  	 11:CASE GVL.mb_Output_Registers[GVL.WATERHARDWARETYPE] OF
(* 		GVL.SWPWTR_TIME:
			//GVL.mb_Output_Registers[GVL.REALTIME_PLC_A2D] :=	0;	//nothing to read with FB circuit, just move motor
			IF GVL.mb_Output_Coils[GVL.REALTIME_ADVANCE] THEN		//move the motor forward
				IF TRUE THEN							//test the FB for limit - can't do this, pass through
					GVL_IO.WaterMotorFwd[FTN1] := TRUE;				// turn on the advance output
					GVL_IO.WaterMotorRvs[FTN1] := FALSE;
					wCycleCount := wCycleCount + 1;
					IF wCycleCount > wMotorTimeOn THEN				//done with timer?
						GVL_IO.WaterMotorFwd[FTN1] := FALSE;		//turn off outputs
						GVL_IO.WaterMotorRvs[FTN1] := FALSE;
						GVL.mb_Output_Coils[GVL.REALTIME_ADVANCE] := FALSE; // reset the advance boolean
						wCycleCount := 0;					//reset the timer counter						
					END_IF
				END_IF
			END_IF
			IF GVL.mb_Output_Coils[GVL.REALTIME_RETARD] THEN
				IF TRUE THEN							//test the FB for limit - can't do this, pass through
					GVL_IO.WaterMotorFwd[FTN1] := FALSE;				// turn on the reverse output
					GVL_IO.WaterMotorRvs[FTN1] := TRUE;
					wCycleCount := wCycleCount + 1;
					IF wCycleCount > wMotorTimeOn THEN				//done with timer?
						GVL_IO.WaterMotorFwd[FTN1] := FALSE;		//turn off outputs
						GVL_IO.WaterMotorRvs[FTN1] := FALSE;
						GVL.mb_Output_Coils[GVL.REALTIME_RETARD] := FALSE; // reset the reverse boolean
						wCycleCount := 0;					//reset the timer counter						
					END_IF
				END_IF
			END_IF
		GVL.SWPWTR_FB:
			GVL.mb_Output_Registers[GVL.REALTIME_PLC_A2D] :=	INT_TO_WORD(GVL_IO.WaterInput[FTN1]);
			IF GVL.mb_Output_Coils[GVL.REALTIME_ADVANCE] THEN		//move the motor forward
				IF GVL_IO.WaterInput[FTN1] < 32000 THEN				//test the FB for limit - assumes 32767 is max of 10 VDC
					GVL_IO.WaterMotorFwd[FTN1] := TRUE;				// turn on the advance output
					GVL_IO.WaterMotorRvs[FTN1] := FALSE;
					wCycleCount := wCycleCount + 1;
					IF wCycleCount > wMotorTimeOn THEN				//done with timer?
						GVL_IO.WaterMotorFwd[FTN1] := FALSE;		//turn off outputs
						GVL_IO.WaterMotorRvs[FTN1] := FALSE;
						GVL.mb_Output_Coils[GVL.REALTIME_ADVANCE] := FALSE; // reset the advance boolean
						wCycleCount := 0;					//reset the timer counter						
						//  curr % sweep   curr ticks - min tick allowed      max sweep %            max ticks allowed      min ticks allowed
						GVL.mb_Output_Registers[GVL.SWEEPTRIMONPRESS + (FTN1 * GVL.WORDRUNTIMEGROUPSIZE)]	:= (INT_TO_WORD(GVL_IO.InkInput[FTN1]) - GVL.w_InkInputIntMin[FTN1]) * 
								(GVL.mb_Output_Registers[GVL.MAXSWEEPTRIM]+1) / (GVL.w_InkInputIntMax[FTN1] - GVL.w_InkInputIntMin[FTN1]);
						//need the onpress setting pointed to the current % sweep of the positioner
					END_IF
				END_IF
			END_IF
			IF GVL.mb_Output_Coils[GVL.REALTIME_RETARD] THEN
				IF GVL_IO.WaterInput[FTN1] > 800 THEN				//test the FB for limit - assumes 32767 is max of 10 VDC
					GVL_IO.WaterMotorFwd[FTN1] := FALSE;				// turn on the reverse output
					GVL_IO.WaterMotorRvs[FTN1] := TRUE;
					wCycleCount := wCycleCount + 1;
					IF wCycleCount > wMotorTimeOn THEN				//done with timer?
						GVL_IO.WaterMotorFwd[FTN1] := FALSE;		//turn off outputs
						GVL_IO.WaterMotorRvs[FTN1] := FALSE;
						GVL.mb_Output_Coils[GVL.REALTIME_RETARD] := FALSE; // reset the reverse boolean
						wCycleCount := 0;					//reset the timer counter						
						//  curr % sweep   curr ticks - min tick allowed      max sweep %            max ticks allowed      min ticks allowed
						GVL.mb_Output_Registers[GVL.SWEEPTRIMONPRESS + (FTN1 * GVL.WORDRUNTIMEGROUPSIZE)]	:= (INT_TO_WORD(GVL_IO.InkInput[FTN1]) - GVL.w_InkInputIntMin[FTN1]) * 
								(GVL.mb_Output_Registers[GVL.MAXSWEEPTRIM]+1) / (GVL.w_InkInputIntMax[FTN1] - GVL.w_InkInputIntMin[FTN1]);
						//need the onpress setting pointed to the current % sweep of the positioner
					END_IF
				END_IF
			END_IF
		GVL.SWPWTR_OUTPUT:
			IF( GVL.b_DINTInput) THEN									//how big should the adv / ret control increment be?
				w_output_incr :=  DINT_TO_INT(GVL.d_DINT10V / 100);
			ELSE
				w_output_incr := (GVL.i_INT10V / 100);
			END_IF
			GVL.mb_Output_Registers[GVL.REALTIME_PLC_A2D] :=	INT_TO_WORD(GVL_IO.WaterSweepOut[FTN1]);
			IF GVL.mb_Output_Coils[GVL.REALTIME_ADVANCE] THEN
				IF GVL_IO.WaterSweepOut[FTN1] < (w_output_incr * 10) THEN
					GVL_IO.WaterSweepOut[FTN1] := GVL_IO.WaterSweepOut[FTN1] + w_output_incr;
				END_IF
				GVL.mb_Output_Coils[GVL.REALTIME_ADVANCE] := FALSE;
			END_IF
			IF GVL.mb_Output_Coils[GVL.REALTIME_RETARD] THEN
				IF GVL_IO.WaterSweepOut[FTN1] > w_output_incr THEN
					GVL_IO.WaterSweepOut[FTN1] := GVL_IO.WaterSweepOut[FTN1] - w_output_incr;
				END_IF
				GVL.mb_Output_Coils[GVL.REALTIME_RETARD] := FALSE;
			END_IF			
 *)
		GVL.SWPWTR_BRIDGE:
		END_CASE
	 12:CASE GVL.mb_Output_Registers[GVL.WATERHARDWARETYPE] OF
(* 		GVL.SWPWTR_TIME:
			//GVL.mb_Output_Registers[GVL.REALTIME_PLC_A2D] :=	0;	//nothing to read with FB circuit, just move motor
			IF GVL.mb_Output_Coils[GVL.REALTIME_ADVANCE] THEN		//move the motor forward
				IF TRUE THEN							//test the FB for limit - can't do this, pass through
					GVL_IO.WaterMotorFwd[FTN2] := TRUE;				// turn on the advance output
					GVL_IO.WaterMotorRvs[FTN2] := FALSE;
					wCycleCount := wCycleCount + 1;
					IF wCycleCount > wMotorTimeOn THEN				//done with timer?
						GVL_IO.WaterMotorFwd[FTN2] := FALSE;		//turn off outputs
						GVL_IO.WaterMotorRvs[FTN2] := FALSE;
						GVL.mb_Output_Coils[GVL.REALTIME_ADVANCE] := FALSE; // reset the advance boolean
						wCycleCount := 0;					//reset the timer counter						
					END_IF
				END_IF
			END_IF
			IF GVL.mb_Output_Coils[GVL.REALTIME_RETARD] THEN
				IF TRUE THEN							//test the FB for limit - can't do this, pass through
					GVL_IO.WaterMotorFwd[FTN2] := FALSE;				// turn on the reverse output
					GVL_IO.WaterMotorRvs[FTN2] := TRUE;
					wCycleCount := wCycleCount + 1;
					IF wCycleCount > wMotorTimeOn THEN				//done with timer?
						GVL_IO.WaterMotorFwd[FTN2] := FALSE;		//turn off outputs
						GVL_IO.WaterMotorRvs[FTN2] := FALSE;
						GVL.mb_Output_Coils[GVL.REALTIME_RETARD] := FALSE; // reset the reverse boolean
						wCycleCount := 0;					//reset the timer counter						
					END_IF
				END_IF
			END_IF
		GVL.SWPWTR_FB:
			GVL.mb_Output_Registers[GVL.REALTIME_PLC_A2D] :=	INT_TO_WORD(GVL_IO.WaterInput[FTN2]);
			IF GVL.mb_Output_Coils[GVL.REALTIME_ADVANCE] THEN		//move the motor forward
				IF GVL_IO.WaterInput[FTN2] < 32000 THEN				//test the FB for limit - assumes 32767 is max of 10 VDC
					GVL_IO.WaterMotorFwd[FTN2] := TRUE;				// turn on the advance output
					GVL_IO.WaterMotorRvs[FTN2] := FALSE;
					wCycleCount := wCycleCount + 1;
					IF wCycleCount > wMotorTimeOn THEN				//done with timer?
						GVL_IO.WaterMotorFwd[FTN2] := FALSE;		//turn off outputs
						GVL_IO.WaterMotorRvs[FTN2] := FALSE;
						GVL.mb_Output_Coils[GVL.REALTIME_ADVANCE] := FALSE; // reset the advance boolean
						wCycleCount := 0;					//reset the timer counter						
						//  curr % sweep   curr ticks - min tick allowed      max sweep %            max ticks allowed      min ticks allowed
						GVL.mb_Output_Registers[GVL.SWEEPTRIMONPRESS + (FTN2 * GVL.WORDRUNTIMEGROUPSIZE)]	:= (INT_TO_WORD(GVL_IO.InkInput[FTN2]) - GVL.w_InkInputIntMin[FTN2]) * 
								(GVL.mb_Output_Registers[GVL.MAXSWEEPTRIM]+1) / (GVL.w_InkInputIntMax[FTN2] - GVL.w_InkInputIntMin[FTN2]);
						//need the onpress setting pointed to the current % sweep of the positioner
					END_IF
				END_IF
			END_IF
			IF GVL.mb_Output_Coils[GVL.REALTIME_RETARD] THEN
				IF GVL_IO.WaterInput[FTN2] > 800 THEN				//test the FB for limit - assumes 32767 is max of 10 VDC
					GVL_IO.WaterMotorFwd[FTN2] := FALSE;				// turn on the reverse output
					GVL_IO.WaterMotorRvs[FTN2] := TRUE;
					wCycleCount := wCycleCount + 1;
					IF wCycleCount > wMotorTimeOn THEN				//done with timer?
						GVL_IO.WaterMotorFwd[FTN2] := FALSE;		//turn off outputs
						GVL_IO.WaterMotorRvs[FTN2] := FALSE;
						GVL.mb_Output_Coils[GVL.REALTIME_RETARD] := FALSE; // reset the reverse boolean
						wCycleCount := 0;					//reset the timer counter						
						//  curr % sweep   curr ticks - min tick allowed      max sweep %            max ticks allowed      min ticks allowed
						GVL.mb_Output_Registers[GVL.SWEEPTRIMONPRESS + (FTN2 * GVL.WORDRUNTIMEGROUPSIZE)]	:= (INT_TO_WORD(GVL_IO.InkInput[FTN2]) - GVL.w_InkInputIntMin[FTN2]) * 
								(GVL.mb_Output_Registers[GVL.MAXSWEEPTRIM]+1) / (GVL.w_InkInputIntMax[FTN2] - GVL.w_InkInputIntMin[FTN2]);
						//need the onpress setting pointed to the current % sweep of the positioner
					END_IF
				END_IF
			END_IF
		GVL.SWPWTR_OUTPUT:
			IF( GVL.b_DINTInput) THEN									//how big should the adv / ret control increment be?
				w_output_incr :=  DINT_TO_INT(GVL.d_DINT10V / 100);
			ELSE
				w_output_incr := (GVL.i_INT10V / 100);
			END_IF
			GVL.mb_Output_Registers[GVL.REALTIME_PLC_A2D] :=	INT_TO_WORD(GVL_IO.WaterSweepOut[FTN2]);
			IF GVL.mb_Output_Coils[GVL.REALTIME_ADVANCE] THEN
				IF GVL_IO.WaterSweepOut[FTN2] < (w_output_incr * 10) THEN
					GVL_IO.WaterSweepOut[FTN2] := GVL_IO.WaterSweepOut[FTN2] + w_output_incr;
				END_IF
				GVL.mb_Output_Coils[GVL.REALTIME_ADVANCE] := FALSE;
			END_IF
			IF GVL.mb_Output_Coils[GVL.REALTIME_RETARD] THEN
				IF GVL_IO.WaterSweepOut[FTN2] > w_output_incr THEN
					GVL_IO.WaterSweepOut[FTN2] := GVL_IO.WaterSweepOut[FTN2] - w_output_incr;
				END_IF
				GVL.mb_Output_Coils[GVL.REALTIME_RETARD] := FALSE;
			END_IF			
 *)
		GVL.SWPWTR_BRIDGE:
		END_CASE
	 13:CASE GVL.mb_Output_Registers[GVL.WATERHARDWARETYPE] OF
(* 		GVL.SWPWTR_TIME:
			//GVL.mb_Output_Registers[GVL.REALTIME_PLC_A2D] :=	0;	//nothing to read with FB circuit, just move motor
			IF GVL.mb_Output_Coils[GVL.REALTIME_ADVANCE] THEN		//move the motor forward
				IF TRUE THEN							//test the FB for limit - can't do this, pass through
					GVL_IO.WaterMotorFwd[FTN3] := TRUE;				// turn on the advance output
					GVL_IO.WaterMotorRvs[FTN3] := FALSE;
					wCycleCount := wCycleCount + 1;
					IF wCycleCount > wMotorTimeOn THEN				//done with timer?
						GVL_IO.WaterMotorFwd[FTN3] := FALSE;		//turn off outputs
						GVL_IO.WaterMotorRvs[FTN3] := FALSE;
						GVL.mb_Output_Coils[GVL.REALTIME_ADVANCE] := FALSE; // reset the advance boolean
						wCycleCount := 0;					//reset the timer counter						
					END_IF
				END_IF
			END_IF
			IF GVL.mb_Output_Coils[GVL.REALTIME_RETARD] THEN
				IF TRUE THEN							//test the FB for limit - can't do this, pass through
					GVL_IO.WaterMotorFwd[FTN3] := FALSE;				// turn on the reverse output
					GVL_IO.WaterMotorRvs[FTN3] := TRUE;
					wCycleCount := wCycleCount + 1;
					IF wCycleCount > wMotorTimeOn THEN				//done with timer?
						GVL_IO.WaterMotorFwd[FTN3] := FALSE;		//turn off outputs
						GVL_IO.WaterMotorRvs[FTN3] := FALSE;
						GVL.mb_Output_Coils[GVL.REALTIME_RETARD] := FALSE; // reset the reverse boolean
						wCycleCount := 0;					//reset the timer counter						
					END_IF
				END_IF
			END_IF
		GVL.SWPWTR_FB:
			GVL.mb_Output_Registers[GVL.REALTIME_PLC_A2D] :=	INT_TO_WORD(GVL_IO.WaterInput[FTN3]);
			IF GVL.mb_Output_Coils[GVL.REALTIME_ADVANCE] THEN		//move the motor forward
				IF GVL_IO.WaterInput[FTN3] < 32000 THEN				//test the FB for limit - assumes 32767 is max of 10 VDC
					GVL_IO.WaterMotorFwd[FTN3] := TRUE;				// turn on the advance output
					GVL_IO.WaterMotorRvs[FTN3] := FALSE;
					wCycleCount := wCycleCount + 1;
					IF wCycleCount > wMotorTimeOn THEN				//done with timer?
						GVL_IO.WaterMotorFwd[FTN3] := FALSE;		//turn off outputs
						GVL_IO.WaterMotorRvs[FTN3] := FALSE;
						GVL.mb_Output_Coils[GVL.REALTIME_ADVANCE] := FALSE; // reset the advance boolean
						wCycleCount := 0;					//reset the timer counter						
						//  curr % sweep   curr ticks - min tick allowed      max sweep %            max ticks allowed      min ticks allowed
						GVL.mb_Output_Registers[GVL.SWEEPTRIMONPRESS + (FTN3 * GVL.WORDRUNTIMEGROUPSIZE)]	:= (INT_TO_WORD(GVL_IO.InkInput[FTN3]) - GVL.w_InkInputIntMin[FTN3]) * 
								(GVL.mb_Output_Registers[GVL.MAXSWEEPTRIM]+1) / (GVL.w_InkInputIntMax[FTN3] - GVL.w_InkInputIntMin[FTN3]);
						//need the onpress setting pointed to the current % sweep of the positioner
					END_IF
				END_IF
			END_IF
			IF GVL.mb_Output_Coils[GVL.REALTIME_RETARD] THEN
				IF GVL_IO.WaterInput[FTN3] > 800 THEN				//test the FB for limit - assumes 32767 is max of 10 VDC
					GVL_IO.WaterMotorFwd[FTN3] := FALSE;				// turn on the reverse output
					GVL_IO.WaterMotorRvs[FTN3] := TRUE;
					wCycleCount := wCycleCount + 1;
					IF wCycleCount > wMotorTimeOn THEN				//done with timer?
						GVL_IO.WaterMotorFwd[FTN3] := FALSE;		//turn off outputs
						GVL_IO.WaterMotorRvs[FTN3] := FALSE;
						GVL.mb_Output_Coils[GVL.REALTIME_RETARD] := FALSE; // reset the reverse boolean
						wCycleCount := 0;					//reset the timer counter						
						//  curr % sweep   curr ticks - min tick allowed      max sweep %            max ticks allowed      min ticks allowed
						GVL.mb_Output_Registers[GVL.SWEEPTRIMONPRESS + (FTN3 * GVL.WORDRUNTIMEGROUPSIZE)]	:= (INT_TO_WORD(GVL_IO.InkInput[FTN3]) - GVL.w_InkInputIntMin[FTN3]) * 
								(GVL.mb_Output_Registers[GVL.MAXSWEEPTRIM]+1) / (GVL.w_InkInputIntMax[FTN3] - GVL.w_InkInputIntMin[FTN3]);
						//need the onpress setting pointed to the current % sweep of the positioner
					END_IF
				END_IF
			END_IF
		GVL.SWPWTR_OUTPUT:
			IF( GVL.b_DINTInput) THEN									//how big should the adv / ret control increment be?
				w_output_incr :=  DINT_TO_INT(GVL.d_DINT10V / 100);
			ELSE
				w_output_incr := (GVL.i_INT10V / 100);
			END_IF
			GVL.mb_Output_Registers[GVL.REALTIME_PLC_A2D] :=	INT_TO_WORD(GVL_IO.WaterSweepOut[FTN3]);
			IF GVL.mb_Output_Coils[GVL.REALTIME_ADVANCE] THEN
				IF GVL_IO.WaterSweepOut[FTN3] < (w_output_incr * 10) THEN
					GVL_IO.WaterSweepOut[FTN3] := GVL_IO.WaterSweepOut[FTN3] + w_output_incr;
				END_IF
				GVL.mb_Output_Coils[GVL.REALTIME_ADVANCE] := FALSE;
			END_IF
			IF GVL.mb_Output_Coils[GVL.REALTIME_RETARD] THEN
				IF GVL_IO.WaterSweepOut[FTN3] > w_output_incr THEN
					GVL_IO.WaterSweepOut[FTN3] := GVL_IO.WaterSweepOut[FTN3] - w_output_incr;
				END_IF
				GVL.mb_Output_Coils[GVL.REALTIME_RETARD] := FALSE;
			END_IF			
 *)
		GVL.SWPWTR_BRIDGE:
		END_CASE
	 14:CASE GVL.mb_Output_Registers[GVL.WATERHARDWARETYPE] OF
(* 		GVL.SWPWTR_TIME:
			//GVL.mb_Output_Registers[GVL.REALTIME_PLC_A2D] :=	0;	//nothing to read with FB circuit, just move motor
			IF GVL.mb_Output_Coils[GVL.REALTIME_ADVANCE] THEN		//move the motor forward
				IF TRUE THEN							//test the FB for limit - can't do this, pass through
					GVL_IO.WaterMotorFwd[FTN4] := TRUE;				// turn on the advance output
					GVL_IO.WaterMotorRvs[FTN4] := FALSE;
					wCycleCount := wCycleCount + 1;
					IF wCycleCount > wMotorTimeOn THEN				//done with timer?
						GVL_IO.WaterMotorFwd[FTN4] := FALSE;		//turn off outputs
						GVL_IO.WaterMotorRvs[FTN4] := FALSE;
						GVL.mb_Output_Coils[GVL.REALTIME_ADVANCE] := FALSE; // reset the advance boolean
						wCycleCount := 0;					//reset the timer counter						
					END_IF
				END_IF
			END_IF
			IF GVL.mb_Output_Coils[GVL.REALTIME_RETARD] THEN
				IF TRUE THEN							//test the FB for limit - can't do this, pass through
					GVL_IO.WaterMotorFwd[FTN4] := FALSE;				// turn on the reverse output
					GVL_IO.WaterMotorRvs[FTN4] := TRUE;
					wCycleCount := wCycleCount + 1;
					IF wCycleCount > wMotorTimeOn THEN				//done with timer?
						GVL_IO.WaterMotorFwd[FTN4] := FALSE;		//turn off outputs
						GVL_IO.WaterMotorRvs[FTN4] := FALSE;
						GVL.mb_Output_Coils[GVL.REALTIME_RETARD] := FALSE; // reset the reverse boolean
						wCycleCount := 0;					//reset the timer counter						
					END_IF
				END_IF
			END_IF
		GVL.SWPWTR_FB:
			GVL.mb_Output_Registers[GVL.REALTIME_PLC_A2D] :=	INT_TO_WORD(GVL_IO.WaterInput[FTN4]);
			IF GVL.mb_Output_Coils[GVL.REALTIME_ADVANCE] THEN		//move the motor forward
				IF GVL_IO.WaterInput[FTN4] < 32000 THEN				//test the FB for limit - assumes 32767 is max of 10 VDC
					GVL_IO.WaterMotorFwd[FTN4] := TRUE;				// turn on the advance output
					GVL_IO.WaterMotorRvs[FTN4] := FALSE;
					wCycleCount := wCycleCount + 1;
					IF wCycleCount > wMotorTimeOn THEN				//done with timer?
						GVL_IO.WaterMotorFwd[FTN4] := FALSE;		//turn off outputs
						GVL_IO.WaterMotorRvs[FTN4] := FALSE;
						GVL.mb_Output_Coils[GVL.REALTIME_ADVANCE] := FALSE; // reset the advance boolean
						wCycleCount := 0;					//reset the timer counter						
						//  curr % sweep   curr ticks - min tick allowed      max sweep %            max ticks allowed      min ticks allowed
						GVL.mb_Output_Registers[GVL.SWEEPTRIMONPRESS + (FTN4 * GVL.WORDRUNTIMEGROUPSIZE)]	:= (INT_TO_WORD(GVL_IO.InkInput[FTN4]) - GVL.w_InkInputIntMin[FTN4]) * 
								(GVL.mb_Output_Registers[GVL.MAXSWEEPTRIM]+1) / (GVL.w_InkInputIntMax[FTN4] - GVL.w_InkInputIntMin[FTN4]);
						//need the onpress setting pointed to the current % sweep of the positioner
					END_IF
				END_IF
			END_IF
			IF GVL.mb_Output_Coils[GVL.REALTIME_RETARD] THEN
				IF GVL_IO.WaterInput[FTN4] > 800 THEN				//test the FB for limit - assumes 32767 is max of 10 VDC
					GVL_IO.WaterMotorFwd[FTN4] := FALSE;				// turn on the reverse output
					GVL_IO.WaterMotorRvs[FTN4] := TRUE;
					wCycleCount := wCycleCount + 1;
					IF wCycleCount > wMotorTimeOn THEN				//done with timer?
						GVL_IO.WaterMotorFwd[FTN4] := FALSE;		//turn off outputs
						GVL_IO.WaterMotorRvs[FTN4] := FALSE;
						GVL.mb_Output_Coils[GVL.REALTIME_RETARD] := FALSE; // reset the reverse boolean
						wCycleCount := 0;					//reset the timer counter						
						//  curr % sweep   curr ticks - min tick allowed      max sweep %            max ticks allowed      min ticks allowed
						GVL.mb_Output_Registers[GVL.SWEEPTRIMONPRESS + (FTN4 * GVL.WORDRUNTIMEGROUPSIZE)]	:= (INT_TO_WORD(GVL_IO.InkInput[FTN4]) - GVL.w_InkInputIntMin[FTN4]) * 
								(GVL.mb_Output_Registers[GVL.MAXSWEEPTRIM]+1) / (GVL.w_InkInputIntMax[FTN4] - GVL.w_InkInputIntMin[FTN4]);
						//need the onpress setting pointed to the current % sweep of the positioner
					END_IF
				END_IF
			END_IF
		GVL.SWPWTR_OUTPUT:
			IF( GVL.b_DINTInput) THEN									//how big should the adv / ret control increment be?
				w_output_incr :=  DINT_TO_INT(GVL.d_DINT10V / 100);
			ELSE
				w_output_incr := (GVL.i_INT10V / 100);
			END_IF
			GVL.mb_Output_Registers[GVL.REALTIME_PLC_A2D] :=	INT_TO_WORD(GVL_IO.WaterSweepOut[FTN4]);
			IF GVL.mb_Output_Coils[GVL.REALTIME_ADVANCE] THEN
				IF GVL_IO.WaterSweepOut[FTN4] < (w_output_incr * 10) THEN
					GVL_IO.WaterSweepOut[FTN4] := GVL_IO.WaterSweepOut[FTN4] + w_output_incr;
				END_IF
				GVL.mb_Output_Coils[GVL.REALTIME_ADVANCE] := FALSE;
			END_IF
			IF GVL.mb_Output_Coils[GVL.REALTIME_RETARD] THEN
				IF GVL_IO.WaterSweepOut[FTN4] > w_output_incr THEN
					GVL_IO.WaterSweepOut[FTN4] := GVL_IO.WaterSweepOut[FTN4] - w_output_incr;
				END_IF
				GVL.mb_Output_Coils[GVL.REALTIME_RETARD] := FALSE;
			END_IF			
 *)
		GVL.SWPWTR_BRIDGE:
		END_CASE
	 15:CASE GVL.mb_Output_Registers[GVL.WATERHARDWARETYPE] OF
(* 		GVL.SWPWTR_TIME:
			//GVL.mb_Output_Registers[GVL.REALTIME_PLC_A2D] :=	0;	//nothing to read with FB circuit, just move motor
			IF GVL.mb_Output_Coils[GVL.REALTIME_ADVANCE] THEN		//move the motor forward
				IF TRUE THEN							//test the FB for limit - can't do this, pass through
					GVL_IO.WaterMotorFwd[FTN5] := TRUE;				// turn on the advance output
					GVL_IO.WaterMotorRvs[FTN5] := FALSE;
					wCycleCount := wCycleCount + 1;
					IF wCycleCount > wMotorTimeOn THEN				//done with timer?
						GVL_IO.WaterMotorFwd[FTN5] := FALSE;		//turn off outputs
						GVL_IO.WaterMotorRvs[FTN5] := FALSE;
						GVL.mb_Output_Coils[GVL.REALTIME_ADVANCE] := FALSE; // reset the advance boolean
						wCycleCount := 0;					//reset the timer counter						
					END_IF
				END_IF
			END_IF
			IF GVL.mb_Output_Coils[GVL.REALTIME_RETARD] THEN
				IF TRUE THEN							//test the FB for limit - can't do this, pass through
					GVL_IO.WaterMotorFwd[FTN5] := FALSE;				// turn on the reverse output
					GVL_IO.WaterMotorRvs[FTN5] := TRUE;
					wCycleCount := wCycleCount + 1;
					IF wCycleCount > wMotorTimeOn THEN				//done with timer?
						GVL_IO.WaterMotorFwd[FTN5] := FALSE;		//turn off outputs
						GVL_IO.WaterMotorRvs[FTN5] := FALSE;
						GVL.mb_Output_Coils[GVL.REALTIME_RETARD] := FALSE; // reset the reverse boolean
						wCycleCount := 0;					//reset the timer counter						
					END_IF
				END_IF
			END_IF
		GVL.SWPWTR_FB:
			GVL.mb_Output_Registers[GVL.REALTIME_PLC_A2D] :=	INT_TO_WORD(GVL_IO.WaterInput[FTN5]);
			IF GVL.mb_Output_Coils[GVL.REALTIME_ADVANCE] THEN		//move the motor forward
				IF GVL_IO.WaterInput[FTN5] < 32000 THEN				//test the FB for limit - assumes 32767 is max of 10 VDC
					GVL_IO.WaterMotorFwd[FTN5] := TRUE;				// turn on the advance output
					GVL_IO.WaterMotorRvs[FTN5] := FALSE;
					wCycleCount := wCycleCount + 1;
					IF wCycleCount > wMotorTimeOn THEN				//done with timer?
						GVL_IO.WaterMotorFwd[FTN5] := FALSE;		//turn off outputs
						GVL_IO.WaterMotorRvs[FTN5] := FALSE;
						GVL.mb_Output_Coils[GVL.REALTIME_ADVANCE] := FALSE; // reset the advance boolean
						wCycleCount := 0;					//reset the timer counter						
						//  curr % sweep   curr ticks - min tick allowed      max sweep %            max ticks allowed      min ticks allowed
						GVL.mb_Output_Registers[GVL.SWEEPTRIMONPRESS + (FTN5 * GVL.WORDRUNTIMEGROUPSIZE)]	:= (INT_TO_WORD(GVL_IO.InkInput[FTN5]) - GVL.w_InkInputIntMin[FTN5]) * 
								(GVL.mb_Output_Registers[GVL.MAXSWEEPTRIM]+1) / (GVL.w_InkInputIntMax[FTN5] - GVL.w_InkInputIntMin[FTN5]);
						//need the onpress setting pointed to the current % sweep of the positioner
					END_IF
				END_IF
			END_IF
			IF GVL.mb_Output_Coils[GVL.REALTIME_RETARD] THEN
				IF GVL_IO.WaterInput[FTN5] > 800 THEN				//test the FB for limit - assumes 32767 is max of 10 VDC
					GVL_IO.WaterMotorFwd[FTN5] := FALSE;				// turn on the reverse output
					GVL_IO.WaterMotorRvs[FTN5] := TRUE;
					wCycleCount := wCycleCount + 1;
					IF wCycleCount > wMotorTimeOn THEN				//done with timer?
						GVL_IO.WaterMotorFwd[FTN5] := FALSE;		//turn off outputs
						GVL_IO.WaterMotorRvs[FTN5] := FALSE;
						GVL.mb_Output_Coils[GVL.REALTIME_RETARD] := FALSE; // reset the reverse boolean
						wCycleCount := 0;					//reset the timer counter						
						//  curr % sweep   curr ticks - min tick allowed      max sweep %            max ticks allowed      min ticks allowed
						GVL.mb_Output_Registers[GVL.SWEEPTRIMONPRESS + (FTN5 * GVL.WORDRUNTIMEGROUPSIZE)]	:= (INT_TO_WORD(GVL_IO.InkInput[FTN5]) - GVL.w_InkInputIntMin[FTN5]) * 
								(GVL.mb_Output_Registers[GVL.MAXSWEEPTRIM]+1) / (GVL.w_InkInputIntMax[FTN5] - GVL.w_InkInputIntMin[FTN5]);
						//need the onpress setting pointed to the current % sweep of the positioner
					END_IF
				END_IF
			END_IF
		GVL.SWPWTR_OUTPUT:
			IF( GVL.b_DINTInput) THEN									//how big should the adv / ret control increment be?
				w_output_incr :=  DINT_TO_INT(GVL.d_DINT10V / 100);
			ELSE
				w_output_incr := (GVL.i_INT10V / 100);
			END_IF
			GVL.mb_Output_Registers[GVL.REALTIME_PLC_A2D] :=	INT_TO_WORD(GVL_IO.WaterSweepOut[FTN5]);
			IF GVL.mb_Output_Coils[GVL.REALTIME_ADVANCE] THEN
				IF GVL_IO.WaterSweepOut[FTN5] < (w_output_incr * 10) THEN
					GVL_IO.WaterSweepOut[FTN5] := GVL_IO.WaterSweepOut[FTN5] + w_output_incr;
				END_IF
				GVL.mb_Output_Coils[GVL.REALTIME_ADVANCE] := FALSE;
			END_IF
			IF GVL.mb_Output_Coils[GVL.REALTIME_RETARD] THEN
				IF GVL_IO.WaterSweepOut[FTN5] > w_output_incr THEN
					GVL_IO.WaterSweepOut[FTN5] := GVL_IO.WaterSweepOut[FTN5] - w_output_incr;
				END_IF
				GVL.mb_Output_Coils[GVL.REALTIME_RETARD] := FALSE;
			END_IF			
 *)
		GVL.SWPWTR_BRIDGE:
		END_CASE
	 16:	CASE GVL.mb_Output_Registers[GVL.WATERHARDWARETYPE] OF
(* 		GVL.SWPWTR_TIME:
			//GVL.mb_Output_Registers[GVL.REALTIME_PLC_A2D] :=	0;	//nothing to read with FB circuit, just move motor
			IF GVL.mb_Output_Coils[GVL.REALTIME_ADVANCE] THEN		//move the motor forward
				IF TRUE THEN							//test the FB for limit - can't do this, pass through
					GVL_IO.WaterMotorFwd[FTN6] := TRUE;				// turn on the advance output
					GVL_IO.WaterMotorRvs[FTN6] := FALSE;
					wCycleCount := wCycleCount + 1;
					IF wCycleCount > wMotorTimeOn THEN				//done with timer?
						GVL_IO.WaterMotorFwd[FTN6] := FALSE;		//turn off outputs
						GVL_IO.WaterMotorRvs[FTN6] := FALSE;
						GVL.mb_Output_Coils[GVL.REALTIME_ADVANCE] := FALSE; // reset the advance boolean
						wCycleCount := 0;					//reset the timer counter						
					END_IF
				END_IF
			END_IF
			IF GVL.mb_Output_Coils[GVL.REALTIME_RETARD] THEN
				IF TRUE THEN							//test the FB for limit - can't do this, pass through
					GVL_IO.WaterMotorFwd[FTN6] := FALSE;				// turn on the reverse output
					GVL_IO.WaterMotorRvs[FTN6] := TRUE;
					wCycleCount := wCycleCount + 1;
					IF wCycleCount > wMotorTimeOn THEN				//done with timer?
						GVL_IO.WaterMotorFwd[FTN6] := FALSE;		//turn off outputs
						GVL_IO.WaterMotorRvs[FTN6] := FALSE;
						GVL.mb_Output_Coils[GVL.REALTIME_RETARD] := FALSE; // reset the reverse boolean
						wCycleCount := 0;					//reset the timer counter						
					END_IF
				END_IF
			END_IF
		GVL.SWPWTR_FB:
			GVL.mb_Output_Registers[GVL.REALTIME_PLC_A2D] :=	INT_TO_WORD(GVL_IO.WaterInput[FTN6]);
			IF GVL.mb_Output_Coils[GVL.REALTIME_ADVANCE] THEN		//move the motor forward
				IF GVL_IO.WaterInput[FTN6] < 32000 THEN				//test the FB for limit - assumes 32767 is max of 10 VDC
					GVL_IO.WaterMotorFwd[FTN6] := TRUE;				// turn on the advance output
					GVL_IO.WaterMotorRvs[FTN6] := FALSE;
					wCycleCount := wCycleCount + 1;
					IF wCycleCount > wMotorTimeOn THEN				//done with timer?
						GVL_IO.WaterMotorFwd[FTN6] := FALSE;		//turn off outputs
						GVL_IO.WaterMotorRvs[FTN6] := FALSE;
						GVL.mb_Output_Coils[GVL.REALTIME_ADVANCE] := FALSE; // reset the advance boolean
						wCycleCount := 0;					//reset the timer counter						
						//  curr % sweep   curr ticks - min tick allowed      max sweep %            max ticks allowed      min ticks allowed
						GVL.mb_Output_Registers[GVL.SWEEPTRIMONPRESS + (FTN6 * GVL.WORDRUNTIMEGROUPSIZE)]	:= (INT_TO_WORD(GVL_IO.InkInput[FTN6]) - GVL.w_InkInputIntMin[FTN6]) * 
								(GVL.mb_Output_Registers[GVL.MAXSWEEPTRIM]+1) / (GVL.w_InkInputIntMax[FTN6] - GVL.w_InkInputIntMin[FTN6]);
						//need the onpress setting pointed to the current % sweep of the positioner
					END_IF
				END_IF
			END_IF
			IF GVL.mb_Output_Coils[GVL.REALTIME_RETARD] THEN
				IF GVL_IO.WaterInput[FTN6] > 800 THEN				//test the FB for limit - assumes 32767 is max of 10 VDC
					GVL_IO.WaterMotorFwd[FTN6] := FALSE;				// turn on the reverse output
					GVL_IO.WaterMotorRvs[FTN6] := TRUE;
					wCycleCount := wCycleCount + 1;
					IF wCycleCount > wMotorTimeOn THEN				//done with timer?
						GVL_IO.WaterMotorFwd[FTN6] := FALSE;		//turn off outputs
						GVL_IO.WaterMotorRvs[FTN6] := FALSE;
						GVL.mb_Output_Coils[GVL.REALTIME_RETARD] := FALSE; // reset the reverse boolean
						wCycleCount := 0;					//reset the timer counter						
						//  curr % sweep   curr ticks - min tick allowed      max sweep %            max ticks allowed      min ticks allowed
						GVL.mb_Output_Registers[GVL.SWEEPTRIMONPRESS + (FTN6 * GVL.WORDRUNTIMEGROUPSIZE)]	:= (INT_TO_WORD(GVL_IO.InkInput[FTN6]) - GVL.w_InkInputIntMin[FTN6]) * 
								(GVL.mb_Output_Registers[GVL.MAXSWEEPTRIM]+1) / (GVL.w_InkInputIntMax[FTN6] - GVL.w_InkInputIntMin[FTN6]);
						//need the onpress setting pointed to the current % sweep of the positioner
					END_IF
				END_IF
			END_IF
		GVL.SWPWTR_OUTPUT:
			IF( GVL.b_DINTInput) THEN									//how big should the adv / ret control increment be?
				w_output_incr :=  DINT_TO_INT(GVL.d_DINT10V / 100);
			ELSE
				w_output_incr := (GVL.i_INT10V / 100);
			END_IF
			GVL.mb_Output_Registers[GVL.REALTIME_PLC_A2D] :=	INT_TO_WORD(GVL_IO.WaterSweepOut[FTN6]);
			IF GVL.mb_Output_Coils[GVL.REALTIME_ADVANCE] THEN
				IF GVL_IO.WaterSweepOut[FTN6] < (w_output_incr * 10) THEN
					GVL_IO.WaterSweepOut[FTN6] := GVL_IO.WaterSweepOut[FTN6] + w_output_incr;
				END_IF
				GVL.mb_Output_Coils[GVL.REALTIME_ADVANCE] := FALSE;
			END_IF
			IF GVL.mb_Output_Coils[GVL.REALTIME_RETARD] THEN
				IF GVL_IO.WaterSweepOut[FTN6] > w_output_incr THEN
					GVL_IO.WaterSweepOut[FTN6] := GVL_IO.WaterSweepOut[FTN6] - w_output_incr;
				END_IF
				GVL.mb_Output_Coils[GVL.REALTIME_RETARD] := FALSE;
			END_IF			
 *)
		GVL.SWPWTR_BRIDGE:
		END_CASE
	 17:CASE GVL.mb_Output_Registers[GVL.WATERHARDWARETYPE] OF
(* 		GVL.SWPWTR_TIME:
			//GVL.mb_Output_Registers[GVL.REALTIME_PLC_A2D] :=	0;	//nothing to read with FB circuit, just move motor
			IF GVL.mb_Output_Coils[GVL.REALTIME_ADVANCE] THEN		//move the motor forward
				IF TRUE THEN							//test the FB for limit - can't do this, pass through
					GVL_IO.WaterMotorFwd[FTN7] := TRUE;				// turn on the advance output
					GVL_IO.WaterMotorRvs[FTN7] := FALSE;
					wCycleCount := wCycleCount + 1;
					IF wCycleCount > wMotorTimeOn THEN				//done with timer?
						GVL_IO.WaterMotorFwd[FTN7] := FALSE;		//turn off outputs
						GVL_IO.WaterMotorRvs[FTN7] := FALSE;
						GVL.mb_Output_Coils[GVL.REALTIME_ADVANCE] := FALSE; // reset the advance boolean
						wCycleCount := 0;					//reset the timer counter						
					END_IF
				END_IF
			END_IF
			IF GVL.mb_Output_Coils[GVL.REALTIME_RETARD] THEN
				IF TRUE THEN							//test the FB for limit - can't do this, pass through
					GVL_IO.WaterMotorFwd[FTN7] := FALSE;				// turn on the reverse output
					GVL_IO.WaterMotorRvs[FTN7] := TRUE;
					wCycleCount := wCycleCount + 1;
					IF wCycleCount > wMotorTimeOn THEN				//done with timer?
						GVL_IO.WaterMotorFwd[FTN7] := FALSE;		//turn off outputs
						GVL_IO.WaterMotorRvs[FTN7] := FALSE;
						GVL.mb_Output_Coils[GVL.REALTIME_RETARD] := FALSE; // reset the reverse boolean
						wCycleCount := 0;					//reset the timer counter						
					END_IF
				END_IF
			END_IF
		GVL.SWPWTR_FB:
			GVL.mb_Output_Registers[GVL.REALTIME_PLC_A2D] :=	INT_TO_WORD(GVL_IO.WaterInput[FTN7]);
			IF GVL.mb_Output_Coils[GVL.REALTIME_ADVANCE] THEN		//move the motor forward
				IF GVL_IO.WaterInput[FTN7] < 32000 THEN				//test the FB for limit - assumes 32767 is max of 10 VDC
					GVL_IO.WaterMotorFwd[FTN7] := TRUE;				// turn on the advance output
					GVL_IO.WaterMotorRvs[FTN7] := FALSE;
					wCycleCount := wCycleCount + 1;
					IF wCycleCount > wMotorTimeOn THEN				//done with timer?
						GVL_IO.WaterMotorFwd[FTN7] := FALSE;		//turn off outputs
						GVL_IO.WaterMotorRvs[FTN7] := FALSE;
						GVL.mb_Output_Coils[GVL.REALTIME_ADVANCE] := FALSE; // reset the advance boolean
						wCycleCount := 0;					//reset the timer counter						
						//  curr % sweep   curr ticks - min tick allowed      max sweep %            max ticks allowed      min ticks allowed
						GVL.mb_Output_Registers[GVL.SWEEPTRIMONPRESS + (FTN7 * GVL.WORDRUNTIMEGROUPSIZE)]	:= (INT_TO_WORD(GVL_IO.InkInput[FTN7]) - GVL.w_InkInputIntMin[FTN7]) * 
								(GVL.mb_Output_Registers[GVL.MAXSWEEPTRIM]+1) / (GVL.w_InkInputIntMax[FTN7] - GVL.w_InkInputIntMin[FTN7]);
						//need the onpress setting pointed to the current % sweep of the positioner
					END_IF
				END_IF
			END_IF
			IF GVL.mb_Output_Coils[GVL.REALTIME_RETARD] THEN
				IF GVL_IO.WaterInput[FTN7] > 800 THEN				//test the FB for limit - assumes 32767 is max of 10 VDC
					GVL_IO.WaterMotorFwd[FTN7] := FALSE;				// turn on the reverse output
					GVL_IO.WaterMotorRvs[FTN7] := TRUE;
					wCycleCount := wCycleCount + 1;
					IF wCycleCount > wMotorTimeOn THEN				//done with timer?
						GVL_IO.WaterMotorFwd[FTN7] := FALSE;		//turn off outputs
						GVL_IO.WaterMotorRvs[FTN7] := FALSE;
						GVL.mb_Output_Coils[GVL.REALTIME_RETARD] := FALSE; // reset the reverse boolean
						wCycleCount := 0;					//reset the timer counter						
						//  curr % sweep   curr ticks - min tick allowed      max sweep %            max ticks allowed      min ticks allowed
						GVL.mb_Output_Registers[GVL.SWEEPTRIMONPRESS + (FTN7 * GVL.WORDRUNTIMEGROUPSIZE)]	:= (INT_TO_WORD(GVL_IO.InkInput[FTN7]) - GVL.w_InkInputIntMin[FTN7]) * 
								(GVL.mb_Output_Registers[GVL.MAXSWEEPTRIM]+1) / (GVL.w_InkInputIntMax[FTN7] - GVL.w_InkInputIntMin[FTN7]);
						//need the onpress setting pointed to the current % sweep of the positioner
					END_IF
				END_IF
			END_IF
		GVL.SWPWTR_OUTPUT:
			IF( GVL.b_DINTInput) THEN									//how big should the adv / ret control increment be?
				w_output_incr :=  DINT_TO_INT(GVL.d_DINT10V / 100);
			ELSE
				w_output_incr := (GVL.i_INT10V / 100);
			END_IF
			GVL.mb_Output_Registers[GVL.REALTIME_PLC_A2D] :=	INT_TO_WORD(GVL_IO.WaterSweepOut[FTN7]);
			IF GVL.mb_Output_Coils[GVL.REALTIME_ADVANCE] THEN
				IF GVL_IO.WaterSweepOut[FTN7] < (w_output_incr * 10) THEN
					GVL_IO.WaterSweepOut[FTN7] := GVL_IO.WaterSweepOut[FTN7] + w_output_incr;
				END_IF
				GVL.mb_Output_Coils[GVL.REALTIME_ADVANCE] := FALSE;
			END_IF
			IF GVL.mb_Output_Coils[GVL.REALTIME_RETARD] THEN
				IF GVL_IO.WaterSweepOut[FTN7] > w_output_incr THEN
					GVL_IO.WaterSweepOut[FTN7] := GVL_IO.WaterSweepOut[FTN7] - w_output_incr;
				END_IF
				GVL.mb_Output_Coils[GVL.REALTIME_RETARD] := FALSE;
			END_IF			
 *)
		GVL.SWPWTR_BRIDGE:
		END_CASE
	 18:CASE GVL.mb_Output_Registers[GVL.WATERHARDWARETYPE] OF
(* 		GVL.SWPWTR_TIME:
			//GVL.mb_Output_Registers[GVL.REALTIME_PLC_A2D] :=	0;	//nothing to read with FB circuit, just move motor
			IF GVL.mb_Output_Coils[GVL.REALTIME_ADVANCE] THEN		//move the motor forward
				IF TRUE THEN							//test the FB for limit - can't do this, pass through
					GVL_IO.WaterMotorFwd[FTN8] := TRUE;				// turn on the advance output
					GVL_IO.WaterMotorRvs[FTN8] := FALSE;
					wCycleCount := wCycleCount + 1;
					IF wCycleCount > wMotorTimeOn THEN				//done with timer?
						GVL_IO.WaterMotorFwd[FTN8] := FALSE;		//turn off outputs
						GVL_IO.WaterMotorRvs[FTN8] := FALSE;
						GVL.mb_Output_Coils[GVL.REALTIME_ADVANCE] := FALSE; // reset the advance boolean
						wCycleCount := 0;					//reset the timer counter						
					END_IF
				END_IF
			END_IF
			IF GVL.mb_Output_Coils[GVL.REALTIME_RETARD] THEN
				IF TRUE THEN							//test the FB for limit - can't do this, pass through
					GVL_IO.WaterMotorFwd[FTN8] := FALSE;				// turn on the reverse output
					GVL_IO.WaterMotorRvs[FTN8] := TRUE;
					wCycleCount := wCycleCount + 1;
					IF wCycleCount > wMotorTimeOn THEN				//done with timer?
						GVL_IO.WaterMotorFwd[FTN8] := FALSE;		//turn off outputs
						GVL_IO.WaterMotorRvs[FTN8] := FALSE;
						GVL.mb_Output_Coils[GVL.REALTIME_RETARD] := FALSE; // reset the reverse boolean
						wCycleCount := 0;					//reset the timer counter						
					END_IF
				END_IF
			END_IF
		GVL.SWPWTR_FB:
			GVL.mb_Output_Registers[GVL.REALTIME_PLC_A2D] :=	INT_TO_WORD(GVL_IO.WaterInput[FTN8]);
			IF GVL.mb_Output_Coils[GVL.REALTIME_ADVANCE] THEN		//move the motor forward
				IF GVL_IO.WaterInput[FTN8] < 32000 THEN				//test the FB for limit - assumes 32767 is max of 10 VDC
					GVL_IO.WaterMotorFwd[FTN8] := TRUE;				// turn on the advance output
					GVL_IO.WaterMotorRvs[FTN8] := FALSE;
					wCycleCount := wCycleCount + 1;
					IF wCycleCount > wMotorTimeOn THEN				//done with timer?
						GVL_IO.WaterMotorFwd[FTN8] := FALSE;		//turn off outputs
						GVL_IO.WaterMotorRvs[FTN8] := FALSE;
						GVL.mb_Output_Coils[GVL.REALTIME_ADVANCE] := FALSE; // reset the advance boolean
						wCycleCount := 0;					//reset the timer counter						
						//  curr % sweep   curr ticks - min tick allowed      max sweep %            max ticks allowed      min ticks allowed
						GVL.mb_Output_Registers[GVL.SWEEPTRIMONPRESS + (FTN8 * GVL.WORDRUNTIMEGROUPSIZE)]	:= (INT_TO_WORD(GVL_IO.InkInput[FTN8]) - GVL.w_InkInputIntMin[FTN8]) * 
								(GVL.mb_Output_Registers[GVL.MAXSWEEPTRIM]+1) / (GVL.w_InkInputIntMax[FTN8] - GVL.w_InkInputIntMin[FTN8]);
						//need the onpress setting pointed to the current % sweep of the positioner
					END_IF
				END_IF
			END_IF
			IF GVL.mb_Output_Coils[GVL.REALTIME_RETARD] THEN
				IF GVL_IO.WaterInput[FTN8] > 800 THEN				//test the FB for limit - assumes 32767 is max of 10 VDC
					GVL_IO.WaterMotorFwd[FTN8] := FALSE;				// turn on the reverse output
					GVL_IO.WaterMotorRvs[FTN8] := TRUE;
					wCycleCount := wCycleCount + 1;
					IF wCycleCount > wMotorTimeOn THEN				//done with timer?
						GVL_IO.WaterMotorFwd[FTN8] := FALSE;		//turn off outputs
						GVL_IO.WaterMotorRvs[FTN8] := FALSE;
						GVL.mb_Output_Coils[GVL.REALTIME_RETARD] := FALSE; // reset the reverse boolean
						wCycleCount := 0;					//reset the timer counter						
						//  curr % sweep   curr ticks - min tick allowed      max sweep %            max ticks allowed      min ticks allowed
						GVL.mb_Output_Registers[GVL.SWEEPTRIMONPRESS + (FTN8 * GVL.WORDRUNTIMEGROUPSIZE)]	:= (INT_TO_WORD(GVL_IO.InkInput[FTN8]) - GVL.w_InkInputIntMin[FTN8]) * 
								(GVL.mb_Output_Registers[GVL.MAXSWEEPTRIM]+1) / (GVL.w_InkInputIntMax[FTN8] - GVL.w_InkInputIntMin[FTN8]);
						//need the onpress setting pointed to the current % sweep of the positioner
					END_IF
				END_IF
			END_IF
		GVL.SWPWTR_OUTPUT:
			IF( GVL.b_DINTInput) THEN									//how big should the adv / ret control increment be?
				w_output_incr :=  DINT_TO_INT(GVL.d_DINT10V / 100);
			ELSE
				w_output_incr := (GVL.i_INT10V / 100);
			END_IF
			GVL.mb_Output_Registers[GVL.REALTIME_PLC_A2D] :=	INT_TO_WORD(GVL_IO.WaterSweepOut[FTN8]);
			IF GVL.mb_Output_Coils[GVL.REALTIME_ADVANCE] THEN
				IF GVL_IO.WaterSweepOut[FTN8] < (w_output_incr * 10) THEN
					GVL_IO.WaterSweepOut[FTN8] := GVL_IO.WaterSweepOut[FTN8] + w_output_incr;
				END_IF
				GVL.mb_Output_Coils[GVL.REALTIME_ADVANCE] := FALSE;
			END_IF
			IF GVL.mb_Output_Coils[GVL.REALTIME_RETARD] THEN
				IF GVL_IO.WaterSweepOut[FTN8] > w_output_incr THEN
					GVL_IO.WaterSweepOut[FTN8] := GVL_IO.WaterSweepOut[FTN8] - w_output_incr;
				END_IF
				GVL.mb_Output_Coils[GVL.REALTIME_RETARD] := FALSE;
			END_IF			
 *)
		GVL.SWPWTR_BRIDGE:
		END_CASE
	 19:CASE GVL.mb_Output_Registers[GVL.WATERHARDWARETYPE] OF
(* 		GVL.SWPWTR_TIME:
			//GVL.mb_Output_Registers[GVL.REALTIME_PLC_A2D] :=	0;	//nothing to read with FB circuit, just move motor
			IF GVL.mb_Output_Coils[GVL.REALTIME_ADVANCE] THEN		//move the motor forward
				IF TRUE THEN							//test the FB for limit - can't do this, pass through
					GVL_IO.WaterMotorFwd[FTN9] := TRUE;				// turn on the advance output
					GVL_IO.WaterMotorRvs[FTN9] := FALSE;
					wCycleCount := wCycleCount + 1;
					IF wCycleCount > wMotorTimeOn THEN				//done with timer?
						GVL_IO.WaterMotorFwd[FTN9] := FALSE;		//turn off outputs
						GVL_IO.WaterMotorRvs[FTN9] := FALSE;
						GVL.mb_Output_Coils[GVL.REALTIME_ADVANCE] := FALSE; // reset the advance boolean
						wCycleCount := 0;					//reset the timer counter						
					END_IF
				END_IF
			END_IF
			IF GVL.mb_Output_Coils[GVL.REALTIME_RETARD] THEN
				IF TRUE THEN							//test the FB for limit - can't do this, pass through
					GVL_IO.WaterMotorFwd[FTN9] := FALSE;				// turn on the reverse output
					GVL_IO.WaterMotorRvs[FTN9] := TRUE;
					wCycleCount := wCycleCount + 1;
					IF wCycleCount > wMotorTimeOn THEN				//done with timer?
						GVL_IO.WaterMotorFwd[FTN9] := FALSE;		//turn off outputs
						GVL_IO.WaterMotorRvs[FTN9] := FALSE;
						GVL.mb_Output_Coils[GVL.REALTIME_RETARD] := FALSE; // reset the reverse boolean
						wCycleCount := 0;					//reset the timer counter						
					END_IF
				END_IF
			END_IF
		GVL.SWPWTR_FB:
			GVL.mb_Output_Registers[GVL.REALTIME_PLC_A2D] :=	INT_TO_WORD(GVL_IO.WaterInput[FTN9]);
			IF GVL.mb_Output_Coils[GVL.REALTIME_ADVANCE] THEN		//move the motor forward
				IF GVL_IO.WaterInput[FTN9] < 32000 THEN				//test the FB for limit - assumes 32767 is max of 10 VDC
					GVL_IO.WaterMotorFwd[FTN9] := TRUE;				// turn on the advance output
					GVL_IO.WaterMotorRvs[FTN9] := FALSE;
					wCycleCount := wCycleCount + 1;
					IF wCycleCount > wMotorTimeOn THEN				//done with timer?
						GVL_IO.WaterMotorFwd[FTN9] := FALSE;		//turn off outputs
						GVL_IO.WaterMotorRvs[FTN9] := FALSE;
						GVL.mb_Output_Coils[GVL.REALTIME_ADVANCE] := FALSE; // reset the advance boolean
						wCycleCount := 0;					//reset the timer counter						
						//  curr % sweep   curr ticks - min tick allowed      max sweep %            max ticks allowed      min ticks allowed
						GVL.mb_Output_Registers[GVL.SWEEPTRIMONPRESS + (FTN9 * GVL.WORDRUNTIMEGROUPSIZE)]	:= (INT_TO_WORD(GVL_IO.InkInput[FTN9]) - GVL.w_InkInputIntMin[FTN9]) * 
								(GVL.mb_Output_Registers[GVL.MAXSWEEPTRIM]+1) / (GVL.w_InkInputIntMax[FTN9] - GVL.w_InkInputIntMin[FTN9]);
						//need the onpress setting pointed to the current % sweep of the positioner
					END_IF
				END_IF
			END_IF
			IF GVL.mb_Output_Coils[GVL.REALTIME_RETARD] THEN
				IF GVL_IO.WaterInput[FTN9] > 800 THEN				//test the FB for limit - assumes 32767 is max of 10 VDC
					GVL_IO.WaterMotorFwd[FTN9] := FALSE;				// turn on the reverse output
					GVL_IO.WaterMotorRvs[FTN9] := TRUE;
					wCycleCount := wCycleCount + 1;
					IF wCycleCount > wMotorTimeOn THEN				//done with timer?
						GVL_IO.WaterMotorFwd[FTN9] := FALSE;		//turn off outputs
						GVL_IO.WaterMotorRvs[FTN9] := FALSE;
						GVL.mb_Output_Coils[GVL.REALTIME_RETARD] := FALSE; // reset the reverse boolean
						wCycleCount := 0;					//reset the timer counter						
						//  curr % sweep   curr ticks - min tick allowed      max sweep %            max ticks allowed      min ticks allowed
						GVL.mb_Output_Registers[GVL.SWEEPTRIMONPRESS + (FTN9 * GVL.WORDRUNTIMEGROUPSIZE)]	:= (INT_TO_WORD(GVL_IO.InkInput[FTN9]) - GVL.w_InkInputIntMin[FTN9]) * 
								(GVL.mb_Output_Registers[GVL.MAXSWEEPTRIM]+1) / (GVL.w_InkInputIntMax[FTN9] - GVL.w_InkInputIntMin[FTN9]);
						//need the onpress setting pointed to the current % sweep of the positioner
					END_IF
				END_IF
			END_IF
		GVL.SWPWTR_OUTPUT:
			IF( GVL.b_DINTInput) THEN									//how big should the adv / ret control increment be?
				w_output_incr :=  DINT_TO_INT(GVL.d_DINT10V / 100);
			ELSE
				w_output_incr := (GVL.i_INT10V / 100);
			END_IF
			GVL.mb_Output_Registers[GVL.REALTIME_PLC_A2D] :=	INT_TO_WORD(GVL_IO.WaterSweepOut[FTN9]);
			IF GVL.mb_Output_Coils[GVL.REALTIME_ADVANCE] THEN
				IF GVL_IO.WaterSweepOut[FTN9] < (w_output_incr * 10) THEN
					GVL_IO.WaterSweepOut[FTN9] := GVL_IO.WaterSweepOut[FTN9] + w_output_incr;
				END_IF
				GVL.mb_Output_Coils[GVL.REALTIME_ADVANCE] := FALSE;
			END_IF
			IF GVL.mb_Output_Coils[GVL.REALTIME_RETARD] THEN
				IF GVL_IO.WaterSweepOut[FTN9] > w_output_incr THEN
					GVL_IO.WaterSweepOut[FTN9] := GVL_IO.WaterSweepOut[FTN9] - w_output_incr;
				END_IF
				GVL.mb_Output_Coils[GVL.REALTIME_RETARD] := FALSE;
			END_IF			
 *)
		GVL.SWPWTR_BRIDGE:
		END_CASE
	 20:CASE GVL.mb_Output_Registers[GVL.WATERHARDWARETYPE] OF
(* 		GVL.SWPWTR_TIME:
			//GVL.mb_Output_Registers[GVL.REALTIME_PLC_A2D] :=	0;	//nothing to read with FB circuit, just move motor
			IF GVL.mb_Output_Coils[GVL.REALTIME_ADVANCE] THEN		//move the motor forward
				IF TRUE THEN							//test the FB for limit - can't do this, pass through
					GVL_IO.WaterMotorFwd[FTN10] := TRUE;				// turn on the advance output
					GVL_IO.WaterMotorRvs[FTN10] := FALSE;
					wCycleCount := wCycleCount + 1;
					IF wCycleCount > wMotorTimeOn THEN				//done with timer?
						GVL_IO.WaterMotorFwd[FTN10] := FALSE;		//turn off outputs
						GVL_IO.WaterMotorRvs[FTN10] := FALSE;
						GVL.mb_Output_Coils[GVL.REALTIME_ADVANCE] := FALSE; // reset the advance boolean
						wCycleCount := 0;					//reset the timer counter						
					END_IF
				END_IF
			END_IF
			IF GVL.mb_Output_Coils[GVL.REALTIME_RETARD] THEN
				IF TRUE THEN							//test the FB for limit - can't do this, pass through
					GVL_IO.WaterMotorFwd[FTN10] := FALSE;				// turn on the reverse output
					GVL_IO.WaterMotorRvs[FTN10] := TRUE;
					wCycleCount := wCycleCount + 1;
					IF wCycleCount > wMotorTimeOn THEN				//done with timer?
						GVL_IO.WaterMotorFwd[FTN10] := FALSE;		//turn off outputs
						GVL_IO.WaterMotorRvs[FTN10] := FALSE;
						GVL.mb_Output_Coils[GVL.REALTIME_RETARD] := FALSE; // reset the reverse boolean
						wCycleCount := 0;					//reset the timer counter						
					END_IF
				END_IF
			END_IF
		GVL.SWPWTR_FB:
			GVL.mb_Output_Registers[GVL.REALTIME_PLC_A2D] :=	INT_TO_WORD(GVL_IO.WaterInput[FTN10]);
			IF GVL.mb_Output_Coils[GVL.REALTIME_ADVANCE] THEN		//move the motor forward
				IF GVL_IO.WaterInput[FTN10] < 32000 THEN				//test the FB for limit - assumes 32767 is max of 10 VDC
					GVL_IO.WaterMotorFwd[FTN10] := TRUE;				// turn on the advance output
					GVL_IO.WaterMotorRvs[FTN10] := FALSE;
					wCycleCount := wCycleCount + 1;
					IF wCycleCount > wMotorTimeOn THEN				//done with timer?
						GVL_IO.WaterMotorFwd[FTN10] := FALSE;		//turn off outputs
						GVL_IO.WaterMotorRvs[FTN10] := FALSE;
						GVL.mb_Output_Coils[GVL.REALTIME_ADVANCE] := FALSE; // reset the advance boolean
						wCycleCount := 0;					//reset the timer counter						
						//  curr % sweep   curr ticks - min tick allowed      max sweep %            max ticks allowed      min ticks allowed
						GVL.mb_Output_Registers[GVL.SWEEPTRIMONPRESS + (FTN10 * GVL.WORDRUNTIMEGROUPSIZE)]	:= (INT_TO_WORD(GVL_IO.InkInput[FTN10]) - GVL.w_InkInputIntMin[FTN10]) * 
								(GVL.mb_Output_Registers[GVL.MAXSWEEPTRIM]+1) / (GVL.w_InkInputIntMax[FTN10] - GVL.w_InkInputIntMin[FTN10]);
						//need the onpress setting pointed to the current % sweep of the positioner
					END_IF
				END_IF
			END_IF
			IF GVL.mb_Output_Coils[GVL.REALTIME_RETARD] THEN
				IF GVL_IO.WaterInput[FTN10] > 800 THEN				//test the FB for limit - assumes 32767 is max of 10 VDC
					GVL_IO.WaterMotorFwd[FTN10] := FALSE;				// turn on the reverse output
					GVL_IO.WaterMotorRvs[FTN10] := TRUE;
					wCycleCount := wCycleCount + 1;
					IF wCycleCount > wMotorTimeOn THEN				//done with timer?
						GVL_IO.WaterMotorFwd[FTN10] := FALSE;		//turn off outputs
						GVL_IO.WaterMotorRvs[FTN10] := FALSE;
						GVL.mb_Output_Coils[GVL.REALTIME_RETARD] := FALSE; // reset the reverse boolean
						wCycleCount := 0;					//reset the timer counter						
						//  curr % sweep   curr ticks - min tick allowed      max sweep %            max ticks allowed      min ticks allowed
						GVL.mb_Output_Registers[GVL.SWEEPTRIMONPRESS + (FTN10 * GVL.WORDRUNTIMEGROUPSIZE)]	:= (INT_TO_WORD(GVL_IO.InkInput[FTN10]) - GVL.w_InkInputIntMin[FTN10]) * 
								(GVL.mb_Output_Registers[GVL.MAXSWEEPTRIM]+1) / (GVL.w_InkInputIntMax[FTN10] - GVL.w_InkInputIntMin[FTN10]);
						//need the onpress setting pointed to the current % sweep of the positioner
					END_IF
				END_IF
			END_IF
		GVL.SWPWTR_OUTPUT:
			IF( GVL.b_DINTInput) THEN									//how big should the adv / ret control increment be?
				w_output_incr :=  DINT_TO_INT(GVL.d_DINT10V / 100);
			ELSE
				w_output_incr := (GVL.i_INT10V / 100);
			END_IF
			GVL.mb_Output_Registers[GVL.REALTIME_PLC_A2D] :=	INT_TO_WORD(GVL_IO.WaterSweepOut[FTN10]);
			IF GVL.mb_Output_Coils[GVL.REALTIME_ADVANCE] THEN
				IF GVL_IO.WaterSweepOut[FTN10] < (w_output_incr * 10) THEN
					GVL_IO.WaterSweepOut[FTN10] := GVL_IO.WaterSweepOut[FTN10] + w_output_incr;
				END_IF
				GVL.mb_Output_Coils[GVL.REALTIME_ADVANCE] := FALSE;
			END_IF
			IF GVL.mb_Output_Coils[GVL.REALTIME_RETARD] THEN
				IF GVL_IO.WaterSweepOut[FTN10] > w_output_incr THEN
					GVL_IO.WaterSweepOut[FTN10] := GVL_IO.WaterSweepOut[FTN10] - w_output_incr;
				END_IF
				GVL.mb_Output_Coils[GVL.REALTIME_RETARD] := FALSE;
			END_IF			
 *)
		GVL.SWPWTR_BRIDGE:
		END_CASE
	 21:   
(*		IF (GVL.b_DINTInput) THEN 
			GVL.mb_Output_Registers[GVL.REALTIME_PLC_A2D] :=	DINT_TO_WORD(GVL_IO.d_PressSpeed/(GVL.d_DINT10V/GVL.i_INT10V))*10;	//press speed (int type)
		ELSE
			GVL.mb_Output_Registers[GVL.REALTIME_PLC_A2D] :=	INT_TO_WORD(GVL_IO.i_PressSpeed);	//press speed (int type)
		END_IF
*)
		GVL.mb_Output_Coils[GVL.REALTIME_ADVANCE] := FALSE; // reset the advance boolean	- no adjustment possible here
		GVL.mb_Output_Coils[GVL.REALTIME_RETARD] := FALSE; // reset the reverse boolean
	 END_CASE

END_FUNCTION_BLOCK

(* stored: Version 1.1.0.1, ProductVersion 3.1.4022.10
   POU FBRealtimeSupport: Id {6abeff8e-f12a-423c-ba2e-ae8ec777e99d}, SpecialFunc None *)
